PROGRAM main
VAR
	CountPulse AT %QX0.0 : bool;
	CountDown AT %QX0.1 : bool;
	ResetCounter AT %QX0.2 : bool;
	Done AT %QX0.3 : bool;
	PartCounter : TF_COUNTER;
	PartCounter_ACC AT %MD0 : DINT;
	PartCounter_OV AT %QX0.4 : BOOL;
	PartCounter_UN AT %QX0.5 : BOOL;
END_VAR

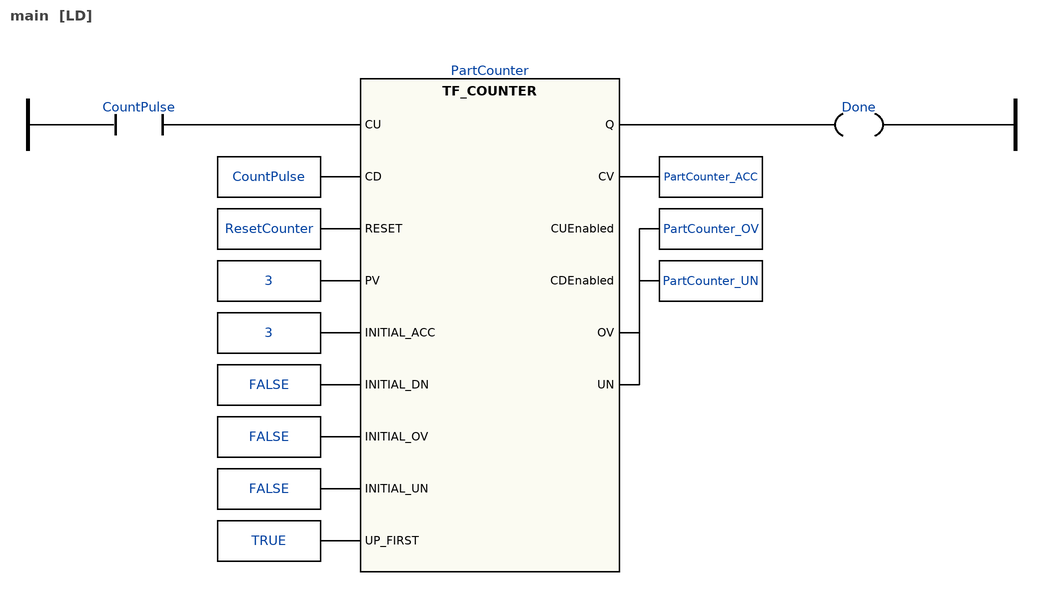
(* LD diagram, written out as Structured Text *)
PartCounter(CU := CountPulse, CD := CountPulse, RESET := ResetCounter, PV := 3, INITIAL_ACC := 3, INITIAL_DN := FALSE, INITIAL_OV := FALSE, INITIAL_UN := FALSE, UP_FIRST := TRUE);
PartCounter_ACC := PartCounter.CV;
PartCounter_OV := PartCounter.OV;
PartCounter_UN := PartCounter.UN;
Done := PartCounter.Q;
END_PROGRAM
